// LS Electric XG5000 project: 동남116
// PLC NewPLC
// module base 0 slot 0: 입출력 모듈:XBC-DN/DP14E (DC 24V 입력 8점, 트랜지스터 출력 6점)

PROGRAM NewProgram (task: 스캔 프로그램)

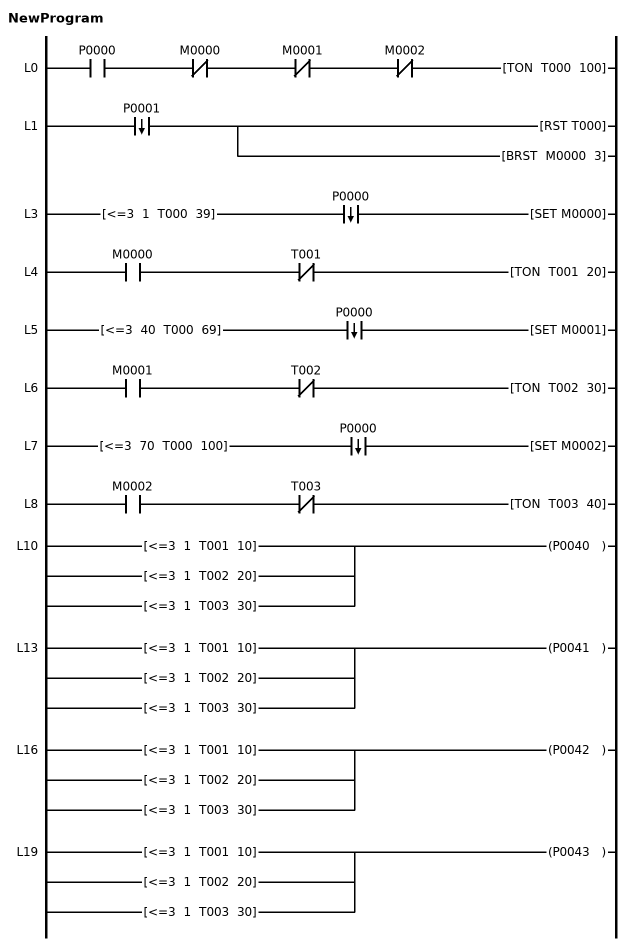
; L0
LOAD      P0000
AND NOT   M0000
AND NOT   M0001
AND NOT   M0002
TON       T000 100
; L1
LOADN     P0001
RST       T000
BRST      M0000 3
; L3
LOAD<=3   1 T000 39
ANDN      P0000
SET       M0000
; L4
LOAD      M0000
AND NOT   T001
TON       T001 20
; L5
LOAD<=3   40 T000 69
ANDN      P0000
SET       M0001
; L6
LOAD      M0001
AND NOT   T002
TON       T002 30
; L7
LOAD<=3   70 T000 100
ANDN      P0000
SET       M0002
; L8
LOAD      M0002
AND NOT   T003
TON       T003 40
; L10
LOAD<=3   1 T001 10
OR<=3     1 T002 20
OR<=3     1 T003 30
OUT       P0040
; L13
LOAD<=3   1 T001 10
OR<=3     1 T002 20
OR<=3     1 T003 30
OUT       P0041
; L16
LOAD<=3   1 T001 10
OR<=3     1 T002 20
OR<=3     1 T003 30
OUT       P0042
; L19
LOAD<=3   1 T001 10
OR<=3     1 T002 20
OR<=3     1 T003 30
OUT       P0043